PROGRAM MAIN
VAR
	Test	: BOOL := FALSE;
	Ready	: BOOL := FALSE;
	i		: INT;
END_VAR


i := i + 1;

IF Ready THEN
	
	Ready := Init();
	
	RETURN;

END_IF


IF Test THEN
	
	Tests();
	
ELSE
	
	Application();
	
END_IF

METHOD Init : BOOL
VAR_INPUT
END_VAR
Init := GVL_EspVisualisation.VisualisationReady;
END_METHOD

END_PROGRAM

(* stored: Version 1.1.0.1
   POU MAIN: Id {85dee3db-2224-4778-955d-df7bd8df7b99}, SpecialFunc None
   Method Init: Id {13e3f36c-2350-4c1a-9b98-cb6bec86661d} *)
